// TIA Portal project "permisos" (V14)

(* hardware
DEVICE "S71500/ET200MP station_1"  S7-1500 station
   slot 0: "Perfil soporte_0"  Rack  6ES7 590-1***0-0AA0
   slot 1: "PLC_2"  CPU 1513-1 PN  6ES7 513-1AL01-0AB0  V2.0
      slot 3: "Display de la CPU_1"  6ES7591-1AA00-0AA0
*)

// ===== PLC "PLC_2"  CPU 1513-1 PN =====

VAR_GLOBAL   // PLC tag table "Tabla de variables estándar"
   "System_Byte" AT %MB1 : Byte;
   "FirstScan" AT %M1.0 : Bool;
   "DiagStatusUpdate" AT %M1.1 : Bool;
   "AlwaysTRUE" AT %M1.2 : Bool;
   "AlwaysFALSE" AT %M1.3 : Bool;
   "Clock_Byte" AT %MB0 : Byte;
   "Clock_10Hz" AT %M0.0 : Bool;
   "Clock_5Hz" AT %M0.1 : Bool;
   "Clock_2.5Hz" AT %M0.2 : Bool;
   "Clock_2Hz" AT %M0.3 : Bool;
   "Clock_1.25Hz" AT %M0.4 : Bool;
   "Clock_1Hz" AT %M0.5 : Bool;
   "Clock_0.625Hz" AT %M0.6 : Bool;
   "Clock_0.5Hz" AT %M0.7 : Bool;
END_VAR

// folder: 1 Valvula

DATA_BLOCK "DB-Valvula"   // DB100
{ S7_Optimized_Access := 'TRUE' }
VERSION : 0.1
   VAR
      Salida : Bool;
      Marcha : Bool;
      Permiso : Bool;
   END_VAR
BEGIN
END_DATA_BLOCK

// folder: 2 Cinta

DATA_BLOCK "DB-Cinta"   // DB200
{ S7_Optimized_Access := 'TRUE' }
VERSION : 0.1
   VAR
      Salida : Bool;
      Marcha : Bool;
      Inductivo : Bool;
      Contaje : Int;
      flkContaje : Bool;
      flkResetContaje : Bool;
   END_VAR
BEGIN
END_DATA_BLOCK

// folder: (top level)

ORGANIZATION_BLOCK "Main"   // OB1, LAD, ProgramCycle
TITLE = "Main Program Sweep (Cycle)"
{ S7_Optimized_Access := 'TRUE' }
VERSION : 0.1
   VAR_INPUT
      Initial_Call : Bool;   // Initial call of this OB
      Remanence : Bool;   // =True, if remanent data are available
   END_VAR
   VAR_TEMP   // added for the SCL form of the ladder/FBD networks
      _w1 : Bool;
   END_VAR
BEGIN

REGION Network 1
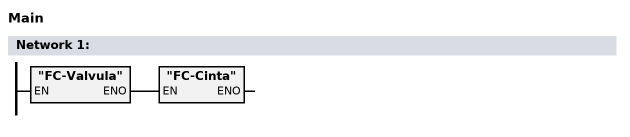
   RUNG wire#powerrail
      "FC-Valvula"()
      "FC-Cinta"()
   END_RUNG
   // the same network as SCL:
   "FC-Valvula"(ENO => #_w1);
   IF #_w1 THEN "FC-Cinta"(); END_IF;
END_REGION
END_ORGANIZATION_BLOCK

// folder: 1 Valvula

FUNCTION "FC-Valvula" : Void   // FC100, LAD
{ S7_Optimized_Access := 'TRUE' }
VERSION : 0.1
BEGIN

REGION Network 1
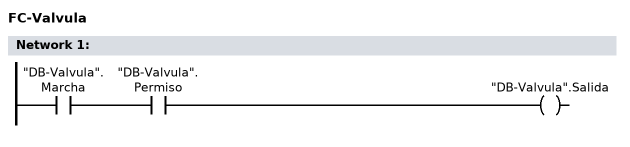
   RUNG wire#powerrail
      Contact( "DB-Valvula".Marcha )
      Contact( "DB-Valvula".Permiso )
      Coil( "DB-Valvula".Salida )
   END_RUNG
   // the same network as SCL:
   "DB-Valvula".Salida := "DB-Valvula".Marcha AND "DB-Valvula".Permiso;
END_REGION
END_FUNCTION

// folder: 2 Cinta

FUNCTION "FC-Cinta" : Void   // FC200, LAD
{ S7_Optimized_Access := 'TRUE' }
VERSION : 0.1
   VAR_TEMP   // added for the SCL form of the ladder/FBD networks
      _w1 : Bool;
      _w2 : Bool;
      _w3 : Bool;
      _w4 : Bool;
   END_VAR
BEGIN

REGION Network 1
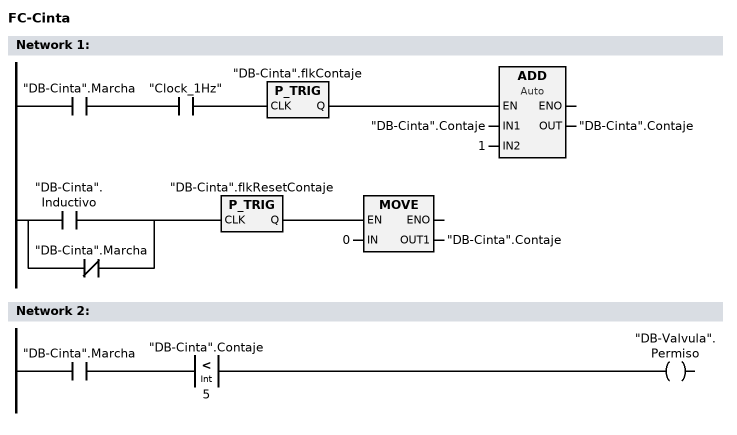
   RUNG wire#powerrail
      Contact( "DB-Cinta".Marcha )
      Contact( "Clock_1Hz" )
      P_Trig( "DB-Cinta".flkContaje )
      Add(in1 := "DB-Cinta".Contaje, in2 := 1, out => "DB-Cinta".Contaje)
   END_RUNG
   RUNG wire#powerrail
      Contact( "DB-Cinta".Inductivo )
      wire#w1
      P_Trig( "DB-Cinta".flkResetContaje )
      Move(in := 0, out1 => "DB-Cinta".Contaje)
   END_RUNG
   RUNG wire#powerrail
      I_Contact( "DB-Cinta".Marcha )
   END_RUNG wire#w1
   // the same network as SCL:
   #_w1 := "DB-Cinta".Marcha AND "Clock_1Hz";
   #_w2 := #_w1 AND NOT "DB-Cinta".flkContaje;   // rising edge
   "DB-Cinta".flkContaje := #_w1;
   IF #_w2 THEN "DB-Cinta".Contaje := "DB-Cinta".Contaje + 1; END_IF;
   #_w3 := "DB-Cinta".Inductivo OR NOT "DB-Cinta".Marcha;
   #_w4 := #_w3 AND NOT "DB-Cinta".flkResetContaje;   // rising edge
   "DB-Cinta".flkResetContaje := #_w3;
   IF #_w4 THEN "DB-Cinta".Contaje := 0; END_IF;
END_REGION

REGION Network 2
   RUNG wire#powerrail
      Contact( "DB-Cinta".Marcha )
      { S7_Templates := "SrcType := Int" } LT_Contact(in1 := "DB-Cinta".Contaje, in2 := 5)
      Coil( "DB-Valvula".Permiso )
   END_RUNG
   // the same network as SCL:
   "DB-Valvula".Permiso := "DB-Cinta".Marcha AND ("DB-Cinta".Contaje < 5);
END_REGION
END_FUNCTION